PROGRAM MAIN
VAR
	
fb_solvexy:FB_SOLVEXY;

END_VAR

GVL.blink := NOT(GVL.blink);

fb_solvexy.x:=GVL.Xc;
fb_solvexy.y:=GVL.Yc;
fb_solvexy();
GVL.alfa:=fb_solvexy.alfa;
GVL.beta:=fb_solvexy.beta;

END_PROGRAM

(* stored: Version 1.1.0.1, ProductVersion 3.1.4024.4
   POU MAIN: Id {d89af4a1-5c9c-4631-9fc2-66e77163c97b}, SpecialFunc None *)
